{attribute 'no_explicit_call' := 'MySingleton is a CLASS and must be accessed using methods or properties'}
FUNCTION_BLOCK MySingleton IMPLEMENTS I_Singleton
VAR 
	singleton					: I_Singleton;	// define the static class instance	
	singletonInstance			: POINTER TO Singleton;
END_VAR

METHOD FB_exit : BOOL
VAR_INPUT
	bInCopyCode : BOOL; // if TRUE, the exit method is called for exiting an instance that is copied afterwards (online change).
END_VAR
// first instance? 
IF singletonInstance <> 0	THEN
	singleton := 0;
	__DELETE(singletonInstance);
	singletonInstance:=0;
END_IF
END_METHOD

METHOD FB_init : BOOL
VAR_INPUT
	bInitRetains : BOOL; // if TRUE, the retain variables are initialized (warm start / cold start)
	bInCopyCode : BOOL;  // if TRUE, the instance afterwards gets moved into the copy code (online change)
END_VAR
// first instance? 
IF singletonInstance = 0	THEN
	singletonInstance := __NEW(Singleton);
	singleton := singletonInstance^;
END_IF
END_METHOD

METHOD FB_reinit : BOOL
VAR_INPUT
END_VAR
__DELETE(singletonInstance);
singleton := 0;
END_METHOD

METHOD Message : STRING
IF singleton <> 0 THEN
	Message := singleton.Message();
END_IF
END_METHOD

END_FUNCTION_BLOCK

(* stored: Version 1.1.0.1, ProductVersion 3.1.4024.11
   POU MySingleton: Id {55dfbb2e-8b31-4adc-9b74-9c9815495848}, SpecialFunc None
   Method FB_exit: Id {89502b3d-46b3-4094-b7c6-c45203e84f2c}
   Method FB_init: Id {225be5fa-b9fe-410e-8547-134eed75cdee}
   Method FB_reinit: Id {834bc95d-6912-4d09-935b-4149d369289a}
   Method Message: Id {b61cfcdd-f85d-4a75-ace3-04e90f0c86cb} *)
